{attribute 'OPC.UA.DA' := '0'}
TYPE Interlock :
STRUCT
	Name : STRING;
	Description : STRING;
	InterlockID : UINT;
	State AT %I* : BOOL;
END_STRUCT
END_TYPE

(* stored: Version 1.1.0.1, ProductVersion 3.1.4024.12
   DUT Interlock: Id {ac16dfdb-9b68-444a-a29e-ef886567bd71} *)
